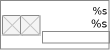
VISUALIZATION VIS_SENSOR_FLAT_RIGHT_MIDDLE  // 110x50
VAR_INPUT
    ITF_SENSOR_IN   :   ITF_SENSOR;	
END_VAR
VAR_INPUT CONSTANT	
	stExklParameter	:	STRING [40] := ' ';	
END_VAR
VAR CONSTANT
	uiIconNr		:	UINT := 2;
END_VAR
    Frame (0,0 110x50), invisible if: NOT fcCheckQuerryAndIconReturn(_ITF_IN := ITF_SENSOR_IN, _uiIconNr_IN := uiIconNr)
        shows VIS_SENSOR_FLAT_RigthMiddleCheckQuerry(ITF_SENSOR_IN := ITF_SENSOR_IN, stExklParameter := stExklParameter)
END_VISUALIZATION

// 40 Visualizations/ICON/SENSOR_FLAT/SENSOR_FLAT_TXT_RIGHT/MIDDLE/VIS_SENSOR_FLAT_RigthMiddleCheckIsEnabled
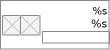
VISUALIZATION VIS_SENSOR_FLAT_RigthMiddleCheckIsEnabled  // 110x50
VAR_INPUT
    ITF_SENSOR_IN   :   ITF_SENSOR;
	stExklParameter	:	STRING [40];	
END_VAR
    Frame (2,15 38x20), invisible if: NOT ITF_SENSOR_IN.proIsEnabled
        shows SensorFlat(ITF_SENSORIN := ITF_SENSOR_IN)
    Frame (42,5 68x40), invisible if: NOT ITF_SENSOR_IN.proIsEnabled
        shows ValueUpDwn(ITF_SENSORIN := ITF_SENSOR_IN, uiTextAusrichtung := 4)
    Rectangle (0,0 110x50)
        OnMouseClick:  Dialog=POPUP_SENSOR, Parameters={stExklParameter: stExklParameter, ITF_SENSORIN: ITF_SENSOR_IN, uiPopUpGruppe: 0}, OpenCentered=True
END_VISUALIZATION

// 40 Visualizations/ICON/SENSOR_FLAT/SENSOR_FLAT_TXT_RIGHT/MIDDLE/VIS_SENSOR_FLAT_RigthMiddleCheckQuerry
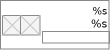
VISUALIZATION VIS_SENSOR_FLAT_RigthMiddleCheckQuerry  // 110x50
VAR_INPUT
    ITF_SENSOR_IN   :   ITF_SENSOR;
	stExklParameter	:	STRING [40];
END_VAR
    Frame (0,0 110x50)
        shows VIS_SENSOR_FLAT_RigthMiddleCheckIsEnabled(ITF_SENSOR_IN := ITF_SENSOR_IN, stExklParameter := stExklParameter)
END_VISUALIZATION

// 40 Visualizations/POPUP/PLACEHOLDER/VIS_SENSOR_PLACEHOLDER
VISUALIZATION VIS_SENSOR_PLACEHOLDER  // 400x400
    Frame (0,0 400x400)
        shows VIS_SENSOR_PLACEHOLDER0()
END_VISUALIZATION

// 40 Visualizations/POPUP/PLACEHOLDER/VIS_SENSOR_PLACEHOLDER0
VISUALIZATION VIS_SENSOR_PLACEHOLDER0  // 400x400
END_VISUALIZATION

// 40 Visualizations/POPUP/PLACEHOLDER/VIS_SENSOR_PLACEHOLDER_1
VISUALIZATION VIS_SENSOR_PLACEHOLDER_1  // 400x400
    Frame (0,0 400x400)
        shows VIS_SENSOR_PLACEHOLDER0_1()
END_VISUALIZATION

// 40 Visualizations/POPUP/PLACEHOLDER/VIS_SENSOR_PLACEHOLDER0_1
VISUALIZATION VIS_SENSOR_PLACEHOLDER0_1  // 400x400
END_VISUALIZATION

(* text list Error (id | default | de | en | fr | it)
  0 | keine Meldung Anstehend | Keine Meldung Anstehend | No message pending | Aucun message en attente | Nessun messaggio in sospeso
  1 | Digital Signal tief | Digital Signal tief | Digital signal low | Signal numérique bas | Segnale digitale basso
  2 | Digital Signal hoch | Digital Signal hoch | Digital signal high | Signal numérique élevé | Segnale digitale alto
  3 | Minimalwert erreicht | Minimalwert erreicht | Minimum value reached | Valeur maximale atteint | Valore massimo raggiunto
  4 | Maximalwert erreicht | Maximalwert erreicht | Maximum value reached | Défaillance de l'interrupteur de protection du moteur | Guasto al salvamotore
  5 | Sensorleitung ist unterbrochen | Sensorleitung ist unterbrochen | sensor line is interrupted | la ligne du capteur est interrompue | La linea del sensore è interrotta
  6 | Sensorleitung hat kurzschluss | Sensorleitung hat kurzschluss | sensor line has overflow | le câble du capteur a un trop-plein | il cavo del sensore ha un trabocco
  7 | Konfigurationsfehler speichern fehlgeschlagen reboot | Konfigurationsfehler speichern fehlgeschlagen reboot | Failed to save configuration error reboot | Impossible d'enregistrer l'erreur de configuration reboot | Impossibile salvare l'errore di configurazione reboot
   |  |  |  |  |  *)

(* text list Info (id | default | de | en | fr | it)
  0 | keine Meldung Anstehend | keine Meldung Anstehend | no message pending | aucun message en attente | nessun messaggio in sospeso
   |  |  |  |  |  *)

(* text list Warnung (id | default | de | en | fr | it)
  0 | Keine Meldung Anstehend | Keine Meldung Anstehend | No message pending | Aucun message en attente | Nessun messaggio in sospeso
  4 | Maximalwert erreicht | Maximalwert erreicht | Maximum value reached | Valeur maximale atteint | Valore massimo raggiunto
  3 | Minimalwert erreicht | Minimalwert erreicht | Minimum value reached | Valeur minimale atteinte | Valore minimo raggiunto
  2 | Digital Signal hoch | Digital Signal hoch | Digital signal high | Signal numérique élevé | Segnale digitale alto
  1 | Digital Signal tief | Digital Signal tief | Digital signal low | Signal numérique bas | Segnale digitale basso
  5 | Wahlschalter Hand, Aus | Wahlschalter Hand, Aus | Selector switch hand off | Commutateur de sélection a main, Éteint | Selettore a mano, spento
  6 | Wahlschalter Hand, Ein | Wahlschalter Hand, Ein | Selector switch hand on | Commutateur de sélection a main, Allumé | Selettore a mano, acceso
  7 | Kabelbruch | Kabelbruch | Cable break | Rupture de câble | Rottura del cavo
  8 | Kurzschluss | Kurzschluss | Short circuit | Court-circuit | Corto circuito
   |  |  |  |  |  *)

(* text list WarnungsStatus (id | default)
  0 | Inaktiv
  1 | Aktiv
   |  *)

(* text list ValueInputType (id | default | de | en | fr | it)
  0 | Default | Default | Default | Défaut | Predefinito
  1 | Analog Input | Analog Input | Analogue input | Entrée analogique | Ingresso analogico
  2 | Digital Input | Digital Input | Digital input | Entrée numérique | Ingresso digitale
  3 | Analog Input (ITF) | Analog Input (ITF) | Analog Input (ITF) | Entrée analogique (ITF) | Ingresso analogico (ITF)
  4 | Digital Input (ITF) | Digital Input (ITF) | Digital Input (ITF) | Entrée numérique (ITF) | Ingresso digitale (ITF)
   |  |  |  |  |  *)
